FUNCTION_BLOCK FB_Vortex_EL3112 IMPLEMENTS I_VolumeFlowSensor
VAR_INPUT
END_VAR
VAR_OUTPUT
END_VAR
VAR								
	//Property Real value
	fVolFlow : REAL;
	//Raw value
	VolFlowRaw AT %I* : INT;
	//Convertion parameters
	m : REAL := 0.00305185071; //Multiplier for convertion
END_VAR

// Volume Flow measurement with Grundfos Vortex sensor

PROPERTY VolumeFlow : REAL
GET
fVolFlow := m * INT_TO_REAL(VolFlowRaw);
VolumeFlow := THIS^.fVolFlow;
END_GET
END_PROPERTY

END_FUNCTION_BLOCK

(* stored: Version 1.1.0.1
   POU FB_Vortex_EL3112: Id {23953ab1-035f-4a94-a17d-2ee96d89fb3e}, SpecialFunc None
   Property VolumeFlow: Id {54670c57-2382-41bd-85d2-98a1c19c6c3b}
   Get Get: Id {7b2ba617-9b10-4aed-bdce-4147aba7112a} *)
